(* One entry in an Mc3AxisParameterLoader table: which NC axis parameter to
   read, and where in the owning axis to store it. *)
TYPE ST_Mc3ParameterBinding :
STRUCT
	ParameterId : Tc3_Mc3Ptp.EAxisParameterId;
	Target		: POINTER TO LREAL;
END_STRUCT
END_TYPE

(* stored: Version 1.1.0.1, ProductVersion 3.1.4026.20
   DUT ST_Mc3ParameterBinding: Id {12b54c59-aa0a-4c3e-a4ef-868528db6db8} *)
